// TIA Portal project "ElevatorAndTurntableSimulator" (V17)
// Vorlageprojekt für das Buch mit Zielsystem S7-1200

(* hardware
DEVICE "S7-1200-Station_1"  S7-1200 Station
   slot 0: "Baugruppenträger_0"  Rack  V1.0
   slot 1: "PLC_1"  CPU 1211C DC/DC/DC  6ES7 211-1AE40-0XB0  V4.1
*)

// ===== PLC "PLC_1"  CPU 1211C DC/DC/DC =====

VAR_GLOBAL   // PLC tag table "Standard-Variablentabelle"
   "ROLL CONVEYOR 1" AT %A0.0 : Bool;
   "STOP" AT %E0.0 : Bool;
   "START" AT %E0.1 : Bool;
   "Tag_4" AT %M0.0 : Bool;
   "Tag_2" AT %M0.1 : Bool;
   "ROLL CONVEYOR 2" AT %Q0.1 : Bool;
   "DIFFUSE SENSOR 1" AT %I0.2 : Bool;
   "TURNTABLE 1 ROLL +" AT %Q0.2 : Bool;
   "TURNTABLE 1 FRONT LIMIT" AT %I0.3 : Bool;
   "TURNTABLE 1 TURN" AT %Q0.3 : Bool;
   "TT 1 LIMIT 90" AT %I0.4 : Bool;
   "DIFFUSE SENSOR 2" AT %I0.5 : Bool;
   "ROLL CONVEYOR 3" AT %Q0.4 : Bool;
   "ELEVATOR 1 RIGHT LIMIT" AT %I0.6 : Bool;
   "ELEVATOR 1 --" AT %Q0.5 : Bool;
   "ELEVATOR 1 LEFT LIMIT" AT %I0.7 : Bool;
   "ELEVATOR 1 UP" AT %Q0.6 : Bool;
END_VAR

FUNCTION "MHJ-PLC-Lab-Function-S71200" : Void   // FC9000, SCL
{ S7_Optimized_Access := 'TRUE' }
VERSION : 0.1
   VAR_TEMP
      rdTimeReturn : Int;
      outputTime : DTL;
      SyncVal : Byte;
      forVal : Int;
      forVal_2 : Int;
      Value : Byte;
   END_VAR
   VAR CONSTANT
      CompVal : Byte := 16#34;
      Value_01 : Byte := 16#11;
      Value_01_DW : DWord := 16#A165_D992;
      Value_02_DW : DWord := 16#58BE_4401;
   END_VAR
BEGIN

   #Value:=PEEK(area := 16#82,
        dbNumber := 0,
        byteOffset := 511);
   #Value := #Value + 1;

   POKE(area := 16#82,
        dbNumber := 0,
        byteOffset := 511,
        value := #Value);

   POKE(area:=16#81,
        dbNumber:=0,
        byteOffset:=1016,
        value:=#Value_01_DW);
   POKE(area := 16#81,
        dbNumber := 0,
        byteOffset := 1020,
        value := #Value_02_DW);

   POKE(area := 16#81,
        dbNumber := 0,
        byteOffset := 511,
        value := B#16#00);

   FOR #forVal := 0 TO 120 DO
       FOR #forVal_2:=0 TO 10 DO
           #rdTimeReturn:=RD_SYS_T(#outputTime);
           #rdTimeReturn := WR_SYS_T(#outputTime);
           #rdTimeReturn := RD_SYS_T(#outputTime);
           #rdTimeReturn := WR_SYS_T(#outputTime);
       END_FOR;
       #SyncVal:= PEEK(area := 16#81,
                      dbNumber := 0,
                      byteOffset := 511);
       IF #SyncVal = #CompVal THEN
          GOTO M_1;
       END_IF;
   END_FOR;
   RETURN;

   M_1:
   POKE(area := 16#81,
        dbNumber := 0,
        byteOffset := 511,
        value := B#16#0);
END_FUNCTION

ORGANIZATION_BLOCK "Main"   // OB1, LAD, ProgramCycle
TITLE = "Main Program Sweep (Cycle)"
{ S7_Optimized_Access := 'TRUE' }
VERSION : 0.1
   VAR_INPUT
      Initial_Call : Bool;   // Initial call of this OB
      Remanence : Bool;   // =True, if remanent data are available
   END_VAR
BEGIN

REGION Network 1: Konnektierungsbaustein für PLC-Lab
   // Im Netzwerk 1 wird der Konnektierungsbaustein für PLC-Lab aufgerufen.
   // Dieser Aufruf darf nicht entfernt werden!
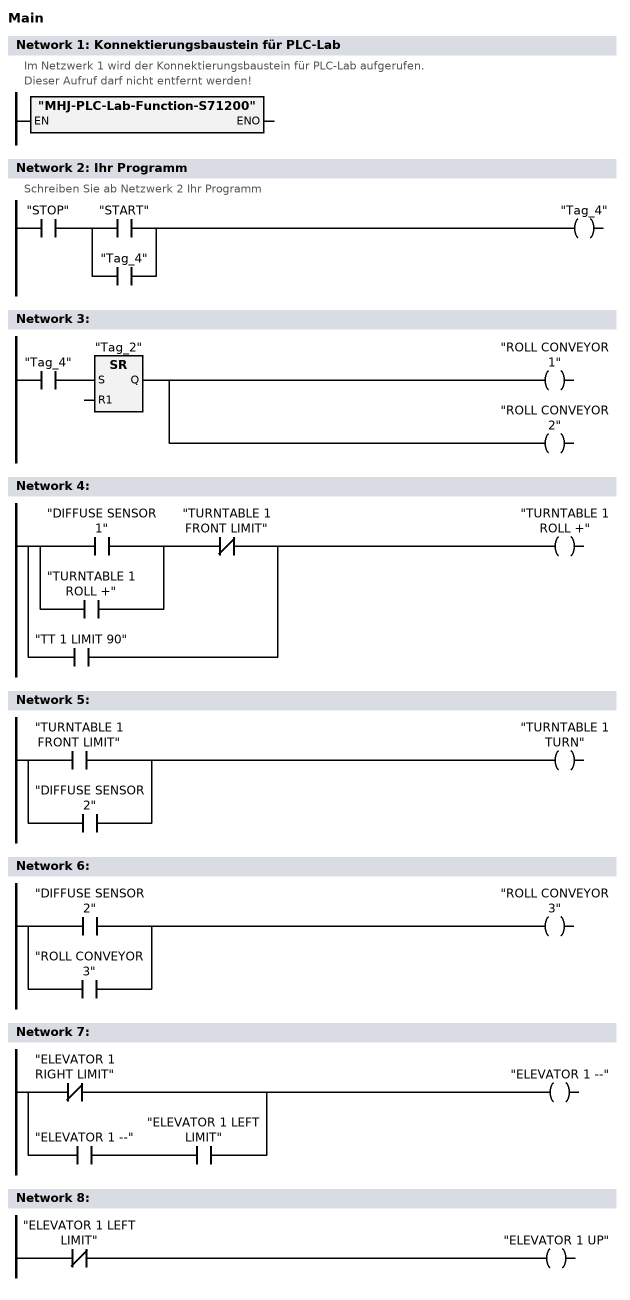
   RUNG wire#powerrail
      "MHJ-PLC-Lab-Function-S71200"()
   END_RUNG
   // the same network as SCL:
   "MHJ-PLC-Lab-Function-S71200"();
END_REGION

REGION Network 2: Ihr Programm
   // Schreiben Sie ab Netzwerk 2 Ihr Programm
   RUNG wire#powerrail
      Contact( "STOP" )
      wire#w1
      Contact( "START" )
      wire#w2
      Coil( "Tag_4" )
   END_RUNG
   RUNG wire#w1
      Contact( "Tag_4" )
   END_RUNG wire#w2
   // the same network as SCL:
   "Tag_4" := "STOP" AND ("START" OR "Tag_4");
END_REGION

REGION Network 3
   RUNG wire#powerrail
      Contact( "Tag_4" )
      S_SR(operand := "Tag_2", r1 :=)
      wire#w1
      Coil( "ROLL CONVEYOR 1" )
   END_RUNG
   RUNG wire#w1
      Coil( "ROLL CONVEYOR 2" )
   END_RUNG
   // the same network as SCL:
   IF "Tag_4" THEN
       "Tag_2" := TRUE;   // SR flip-flop
   END_IF;
   "ROLL CONVEYOR 1" := "Tag_2";
   "ROLL CONVEYOR 2" := "Tag_2";
END_REGION

REGION Network 4
   RUNG wire#powerrail
      Contact( "DIFFUSE SENSOR 1" )
      wire#w1
      I_Contact( "TURNTABLE 1 FRONT LIMIT" )
      wire#w2
      Coil( "TURNTABLE 1 ROLL +" )
   END_RUNG
   RUNG wire#powerrail
      Contact( "TURNTABLE 1 ROLL +" )
   END_RUNG wire#w1
   RUNG wire#powerrail
      Contact( "TT 1 LIMIT 90" )
   END_RUNG wire#w2
   // the same network as SCL:
   "TURNTABLE 1 ROLL +" := (("DIFFUSE SENSOR 1" OR "TURNTABLE 1 ROLL +") AND NOT "TURNTABLE 1 FRONT LIMIT") OR "TT 1 LIMIT 90";
END_REGION

REGION Network 5
   RUNG wire#powerrail
      Contact( "TURNTABLE 1 FRONT LIMIT" )
      wire#w1
      Coil( "TURNTABLE 1 TURN" )
   END_RUNG
   RUNG wire#powerrail
      Contact( "DIFFUSE SENSOR 2" )
   END_RUNG wire#w1
   // the same network as SCL:
   "TURNTABLE 1 TURN" := "TURNTABLE 1 FRONT LIMIT" OR "DIFFUSE SENSOR 2";
END_REGION

REGION Network 6
   RUNG wire#powerrail
      Contact( "DIFFUSE SENSOR 2" )
      wire#w1
      Coil( "ROLL CONVEYOR 3" )
   END_RUNG
   RUNG wire#powerrail
      Contact( "ROLL CONVEYOR 3" )
   END_RUNG wire#w1
   // the same network as SCL:
   "ROLL CONVEYOR 3" := "DIFFUSE SENSOR 2" OR "ROLL CONVEYOR 3";
END_REGION

REGION Network 7
   RUNG wire#powerrail
      I_Contact( "ELEVATOR 1 RIGHT LIMIT" )
      wire#w1
      Coil( "ELEVATOR 1 --" )
   END_RUNG
   RUNG wire#powerrail
      Contact( "ELEVATOR 1 --" )
      Contact( "ELEVATOR 1 LEFT LIMIT" )
   END_RUNG wire#w1
   // the same network as SCL:
   "ELEVATOR 1 --" := NOT "ELEVATOR 1 RIGHT LIMIT" OR ("ELEVATOR 1 --" AND "ELEVATOR 1 LEFT LIMIT");
END_REGION

REGION Network 8
   RUNG wire#powerrail
      I_Contact( "ELEVATOR 1 LEFT LIMIT" )
      Coil( "ELEVATOR 1 UP" )
   END_RUNG
   // the same network as SCL:
   "ELEVATOR 1 UP" := NOT "ELEVATOR 1 LEFT LIMIT";
END_REGION
END_ORGANIZATION_BLOCK